{attribute 'linkalways'} 
{attribute 'no_explicit_call' := 'This FB is a CLASS and must be accessed using methods or properties'}
{attribute 'enable_dynamic_creation'}
FUNCTION_BLOCK ABSTRACT IntegerDatatypeBase EXTENDS DatatypeBase IMPLEMENTS I_IntegerDatatype
VAR
END_VAR

PROPERTY PUBLIC ABSTRACT IsSigned : BOOL
GET
END_GET
END_PROPERTY

METHOD PROTECTED OnSerializeTypeWith
VAR_INPUT
	Serializer : I_Serializer;
END_VAR
SUPER^.OnSerializeTypeWith(Serializer);
Serializer.AddKey('lowerBound');
SerializeLowerbound(Serializer);
Serializer.AddKey('upperBound');
SerializeUpperbound(Serializer);
Serializer.AddKeyBool('isSigned', IsSigned);
END_METHOD

METHOD PROTECTED ABSTRACT SerializeLowerbound
VAR_INPUT
	Serializer : I_Serializer;
END_VAR
END_METHOD

METHOD PROTECTED ABSTRACT SerializeUpperbound
VAR_INPUT
	Serializer : I_Serializer;
END_VAR
END_METHOD

END_FUNCTION_BLOCK

(* stored: Version 1.1.0.1, ProductVersion 3.1.4024.12
   POU IntegerDatatypeBase: Id {6f1eb65d-2dc0-0d58-2e25-2f05b19a5b4c}, SpecialFunc None
   Folder Protected: Id {0775aeec-e6e3-08c0-0bd5-a96fc0b17e35}
   Property IsSigned: Id {eccdeb6f-91bd-0b7e-06bd-f859c210b3de}
   Get Get: Id {1a391de6-e72b-01a7-223d-b1c7d4dcaf6f}
   Method OnSerializeTypeWith: Id {a12cac12-4b78-0363-1a58-b29135d476e6}
   Method SerializeLowerbound: Id {1b3e5609-1076-02ab-1243-ce942263068f}
   Method SerializeUpperbound: Id {0322eecc-293c-0cb4-04c5-f0383a842e65} *)
